Universal Robots PolyScope program: gripper automatico.urp

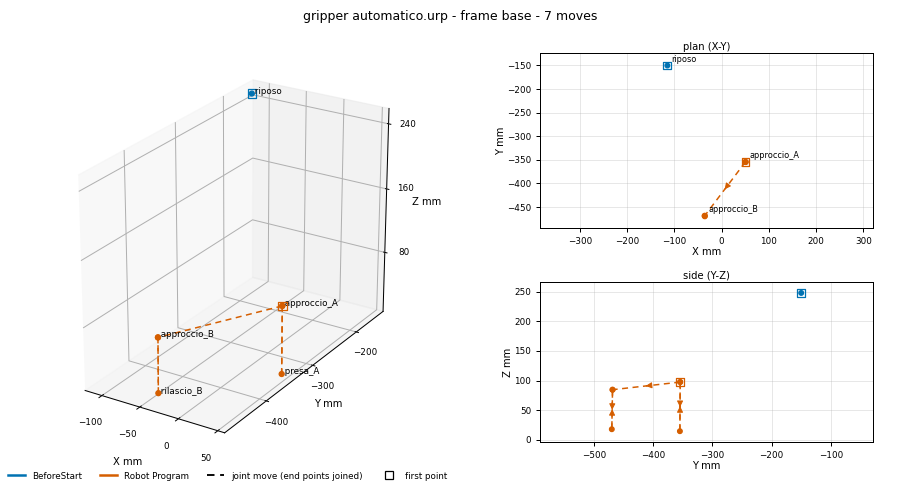
[picture p0: tool path of gripper automatico.urp in frame base, 7 of 7 moves have a stored position in this frame; points joined in program order, loops and branches not executed]
Program gripper automatico (installation=default directory=/programs createdIn=3.15.8.106339 lastSavedIn=3.15.8.106339 robotSerialNumber=2021330429)
Calibrated DH parameters: a=[-0.000156, -0.236402, -0.171625, 0.000006, -0.000047, 0]; d=[0.151683, 29.702709, 78.973085, -108.563557, 0.085229, 0.082167]; alpha=[1.57015, 0.001987, 0.001164, 1.571718, -1.571778, 0]; deltaTheta=[-0.000066, 0.24449, 0.39032, -0.635025, 0.000068, -0.000043]
BeforeStart
  pezzo := False
  URCap Gripper Activate (Robotiq_Grippers, Robotiq Inc.) dataModel(ResetAndActivateKey=false)
  URCap Gripper (Robotiq_Grippers, Robotiq Inc.) dataModel(position=0.0, force=0.0, speed=0.0, positionInDouble=0.0, forceInDouble=0.0, speedInDouble=0.0, slaveIds=[9], blocking=true)
  MoveJ speed 60 deg/s, acceleration 80 deg/s^2 (useActiveTCP=true)
    Waypoint riposo: TCP in base x=-114.781 y=-150.308 z=247.666 mm, rx=2.2629 ry=-1.6199 rz=0.2588 rad; joints [281.971, -35.444, -101.804, -111.371, 82.575, 261.691] deg; flange x=-106.708 y=-90.778 z=392.718 mm, rx=2.2629 ry=-1.6199 rz=0.2588 rad
Robot Program (runOnlyOnce=false)
  MoveJ speed 60 deg/s, acceleration 80 deg/s^2 (useActiveTCP=true)
    Waypoint approccio_A: TCP in base x=50.584 y=-354.333 z=97.612 mm, rx=-2.7944 ry=1.3969 rz=0.0071 rad; joints [296.039, -102.421, -91.676, -76.65, 90.728, 259.067] deg; flange x=49.991 y=-357.104 z=254.587 mm, rx=-2.7944 ry=1.3969 rz=0.0071 rad
    Waypoint presa_A: TCP in base x=50.807 y=-354.77 z=14.621 mm, rx=-2.7962 ry=1.3973 rz=0.0037 rad; joints [296.04, -110.751, -105.174, -54.662, 90.746, 259.077] deg; flange x=50.035 y=-357.147 z=171.601 mm, rx=-2.7962 ry=1.3973 rz=0.0037 rad
    URCap Gripper (Robotiq_Grippers, Robotiq Inc.) dataModel(position=100.0, force=0.0, speed=0.0, positionInDouble=100.0, forceInDouble=0.0, speedInDouble=0.0, slaveIds=[9], blocking=true)
    pezzo := False
    Loop While (checkContinuously=false) expression=pezzo≟ False
      URCap Grip Check (Robotiq_Grippers, Robotiq Inc.) dataModel(DimensionKey=100.0, DimensionDimensionPositiveGapKey=5.0, DimensionNegativeGapKey=5.0, GripperIdKey=1, ModelDefinedKey=true, ObjectDetectedKey=false, DimensionValidationKey=false); state(isChildrenLocked=true)
        URCap If (Robotiq_Grippers, Robotiq Inc.)
          URCap Gripper (Robotiq_Grippers, Robotiq Inc.) dataModel(position=0.0, force=0.0, speed=0.0, positionInDouble=0.0, forceInDouble=0.0, speedInDouble=0.0, slaveIds=[9], blocking=true)
          Wait Sleep waitTime=5
          URCap Gripper (Robotiq_Grippers, Robotiq Inc.) dataModel(position=100.0, force=0.0, speed=0.0, positionInDouble=100.0, forceInDouble=0.0, speedInDouble=0.0, slaveIds=[9], blocking=true)
        URCap Else (Robotiq_Grippers, Robotiq Inc.)
          pezzo := True
    Waypoint uscita_A: TCP in base x=50.515 y=-354.221 z=97.428 mm, rx=-2.7941 ry=1.3968 rz=0.0078 rad; joints [296.038, -102.432, -91.698, -76.651, 90.726, 259.069] deg; flange x=49.969 y=-357.075 z=254.401 mm, rx=-2.7941 ry=1.3968 rz=0.0078 rad
    Waypoint approccio_B: TCP in base x=-35.783 y=-468.303 z=84.556 mm, rx=-2.2412 ry=2.1151 rz=0.0245 rad; joints [278.406, -134.903, -44.318, -93.551, 92.265, 274.947] deg; flange x=-40.413 y=-476.837 z=241.256 mm, rx=-2.2412 ry=2.1151 rz=0.0245 rad
    Waypoint rilascio_B: TCP in base x=-35.617 y=-469.549 z=17.946 mm, rx=-2.2444 ry=2.1178 rz=0.0164 rad; joints [278.409, -137.369, -58.049, -76.973, 92.283, 274.966] deg; flange x=-40.406 y=-477.054 z=174.694 mm, rx=-2.2444 ry=2.1178 rz=0.0164 rad
    URCap Gripper (Robotiq_Grippers, Robotiq Inc.) dataModel(position=0.0, force=0.0, speed=0.0, positionInDouble=0.0, forceInDouble=0.0, speedInDouble=0.0, slaveIds=[9], blocking=true)
    Waypoint uscita_B: TCP in base x=-35.767 y=-468.312 z=84.562 mm, rx=-2.2412 ry=2.1151 rz=0.0244 rad; joints [278.407, -134.903, -44.318, -93.548, 92.267, 274.948] deg; flange x=-40.404 y=-476.839 z=241.262 mm, rx=-2.2412 ry=2.1151 rz=0.0244 rad
